TYPE ST_P_START_OP :
STRUCT
	SetIndex:				BOOl;
	Index:					INT;
	Barcode:				INT;
END_STRUCT
END_TYPE

(* stored: Version 1.1.0.1, ProductVersion 3.1.4024.10
   DUT ST_P_START_OP: Id {83065270-b682-49b5-8d06-ad10db2c3d92} *)
